Universal Robots PolyScope program: test approach.urp

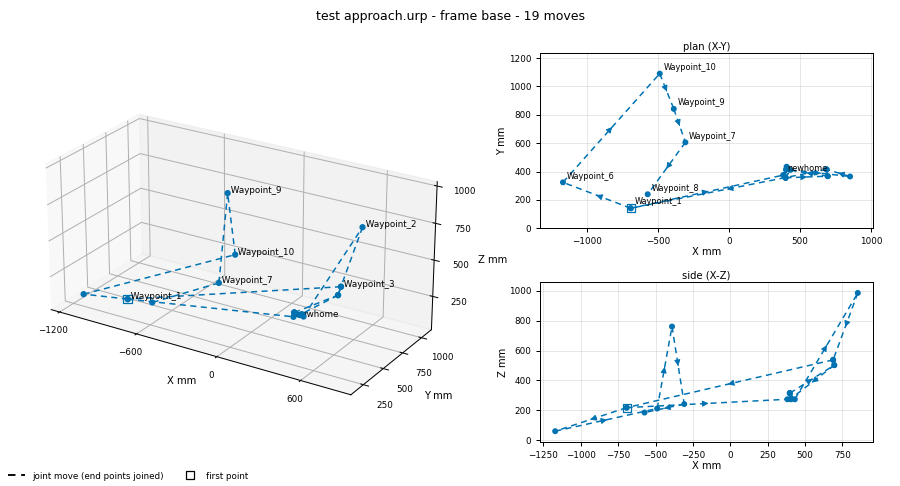
[picture p0: tool path of test approach.urp in frame base, 19 of 19 moves have a stored position in this frame; points joined in program order, loops and branches not executed]
Program test approach (installation=default directory=/programs createdIn=5.14.5 lastSavedIn=5.14.5 robotSerialNumber=20236801216)
Calibrated DH parameters: a=[-0.000021, -0.748897, -0.28186, -0.00004, -0.000055, 0]; d=[0.236225, -424.082933, -1564.66872, 1988.95162, 0.159094, 0.153873]; alpha=[1.570844, 0.001002, 0.000337, 1.571488, -1.569996, 0]; deltaTheta=[0, -0.516316, 5.626292, 1.173211, 0.000001, 0]
InitVariablesNode
Robot Program (runOnlyOnce=false)
  'this program details the steps to get from the old home to the new home'
  SuppressedNode
    SafeHome (positionOptionType=SPEED_AND_ACCELERATION speed=1.047198 acceleration=1.396263 nextMotionTime=2)
  MoveJ speed 60 deg/s, acceleration 80 deg/s^2 (useActiveTCP=true positionType=JointAngles) feature=Base
    Waypoint Waypoint_1: TCP in base x=-693.756 y=141.369 z=218.585 mm, rx=-0.852 ry=-1.646 rz=1.646 rad; joints [-66.082, -85.509, 163.4, 282.028, -281.373, 90.065] deg; TCP offset x=-5.492 y=-332.581 z=106.393 mm, rx=1.2092 ry=-1.2092 rz=1.2092 rad
    Waypoint newhome: TCP in base x=381.329 y=374.762 z=274.442 mm, rx=3.0086 ry=0.1175 rz=0.0082 rad; joints [-134.647, -110.577, 133.203, 337.299, -229.171, -7.533] deg
    Waypoint newhome_face_sa: TCP in base x=405.677 y=434.282 z=274.451 mm, rx=2.2921 ry=2.0938 rz=-0.0024 rad; joints [-182.247, -105.299, 130.564, 360.94, -356.728, -27.679] deg
    Waypoint oldhome: TCP in base x=397.684 y=356.251 z=315.247 mm, rx=2.3163 ry=2.0576 rz=0.0741 rad; joints [-198.127, -117.852, 133.304, -13.011, -11.422, -6.036] deg
  SuppressedNode
    MoveL speed 250 mm/s, acceleration 1200 mm/s^2 (useActiveTCP=true) feature=Base
      Waypoint oldhome: TCP in base x=397.684 y=356.251 z=315.247 mm, rx=2.3163 ry=2.0576 rz=0.0741 rad; joints [-198.127, -117.852, 133.304, -13.011, -11.422, -6.036] deg
      Waypoint newhome_face_sa: TCP in base x=405.677 y=434.282 z=274.451 mm, rx=2.2921 ry=2.0938 rz=-0.0024 rad; joints [-182.247, -105.299, 130.564, 360.94, -356.728, -27.679] deg
      Waypoint newhome_face_nr: TCP in base x=431.376 y=411.557 z=274.165 mm, rx=2.4165 ry=1.9889 rz=0.0007 rad; joints [-186.179, -111.083, 133.075, 342.194, -355.119, -4.712] deg
  MoveJ speed 60 deg/s, acceleration 80 deg/s^2 (useActiveTCP=true positionType=JointAngles) feature=Base
    Waypoint newhome_face_nr: TCP in base x=431.376 y=411.557 z=274.165 mm, rx=2.4165 ry=1.9889 rz=0.0007 rad; joints [-186.179, -111.083, 133.075, 342.194, -355.119, -4.712] deg
    Waypoint Waypoint_2: TCP in base x=852.538 y=365.246 z=985.645 mm, rx=0.9717 ry=0.7885 rz=1.357 rad; joints [-186.178, -111.084, 133.075, 228.144, -355.119, -4.712] deg
    Waypoint Waypoint_3: TCP in base x=687.528 y=415.166 z=537.921 mm, rx=2.1271 ry=1.9299 rz=0.4701 rad; joints [-186.178, -111.085, 133.077, 228.144, -355.12, 87.586] deg
    Waypoint Waypoint_4: TCP in base x=695.155 y=367.452 z=502.522 mm, rx=2.0931 ry=1.8575 rz=0.3088 rad; joints [-186.178, -111.085, 133.076, 228.143, -3.264, 87.587] deg
    Waypoint Waypoint_5: TCP in base x=400.807 y=414.191 z=275.291 mm, rx=2.3676 ry=2.0272 rz=0.0088 rad; joints [-186.175, -111.083, 133.204, -9.066, 2.731, -14.326] deg
    Waypoint oldhome: TCP in base x=397.684 y=356.251 z=315.247 mm, rx=2.3163 ry=2.0576 rz=0.0741 rad; joints [-198.127, -117.852, 133.304, -13.011, -11.422, -6.036] deg
  MoveJ speed 60 deg/s, acceleration 80 deg/s^2 (useActiveTCP=true) feature=Base
    Waypoint oldhome: TCP in base x=397.684 y=356.251 z=315.247 mm, rx=2.3163 ry=2.0576 rz=0.0741 rad; joints [-198.127, -117.852, 133.304, -13.011, -11.422, -6.036] deg
    Waypoint Waypoint_4: TCP in base x=695.155 y=367.452 z=502.522 mm, rx=2.0931 ry=1.8575 rz=0.3088 rad; joints [-186.178, -111.085, 133.076, 228.143, -3.264, 87.587] deg
    Waypoint Waypoint_3: TCP in base x=687.528 y=415.166 z=537.921 mm, rx=2.1271 ry=1.9299 rz=0.4701 rad; joints [-186.178, -111.085, 133.077, 228.144, -355.12, 87.586] deg
    SuppressedNode
      Waypoint Waypoint_2: TCP in base x=852.538 y=365.246 z=985.645 mm, rx=0.9717 ry=0.7885 rz=1.357 rad; joints [-186.178, -111.084, 133.075, 228.144, -355.119, -4.712] deg
    Waypoint Waypoint_1: TCP in base x=-693.756 y=141.369 z=218.585 mm, rx=-0.852 ry=-1.646 rz=1.646 rad; joints [-66.082, -85.509, 163.4, 282.028, -281.373, 90.065] deg
  'approach for right weld in between 2 and 3'
  MoveJ speed 60 deg/s, acceleration 80 deg/s^2 (useActiveTCP=true) feature=Base
    Waypoint Waypoint_6: TCP in base x=-1171.716 y=324.078 z=60.781 mm, rx=0.4204 ry=-1.583 rz=0.541 rad; joints [-41.063, -22.166, 108.862, 188.889, -270.902, 75.98] deg; TCP offset x=6.62 y=-330.62 z=102.07 mm, rx=1.2092 ry=-1.2092 rz=1.2092 rad
    Waypoint Waypoint_10: TCP in base x=-489.526 y=1090.477 z=212.437 mm, rx=-1.9326 ry=-1.3431 rz=1.4553 rad; joints [-90.17, -61.333, 93.006, 0.399, 90.423, 62.4] deg
    Waypoint Waypoint_9: TCP in base x=-390.34 y=842.096 z=760.827 mm, rx=-0.1817 ry=0.0752 rz=-2.9995 rad; joints [-91.332, -61.478, 100.843, -3.085, -11.522, 140.93] deg
    Waypoint Waypoint_7: TCP in base x=-308.539 y=606.07 z=242.399 mm, rx=1.3699 ry=1.0669 rz=-1.2572 rad; joints [-85.579, -53.078, 88.71, 54.847, 94.978, 13.63] deg
    ''
    Waypoint Waypoint_8: TCP in base x=-574.227 y=239.847 z=185.455 mm, rx=1.8953 ry=0.4806 rz=-1.8249 rad; joints [-76.459, -71.594, 130.091, 35.922, 92.316, 70.191] deg
